PROGRAM F_VELOCIDADES
VAR_INPUT
	Func:E_Funcio;
END_VAR
VAR
	///Activa
	xActv: BOOL;
	///Parametros
	wP_SP_SpeedPumpC: WORD;
	wP_SP_Speed: WORD;
	wP_SP_T_Pass: WORD;
	///Fin Funcion
	xFinFunc: BOOL;
	tFinFuncion: Ton;
	a: INT;
	rOutAnalogSpeedPumpC: REAL;
END_VAR


a:=a+1;

(*Activa funcio *)
xActv:= func.Actv_Funcio;

wP_SP_SpeedPumpC:= func.ParamFunc[1];
wP_SP_Speed:= func.ParamFunc[2];
wP_SP_T_Pass:= func.ParamFunc[3];

(*
IF xActv
	THEN
	(*Torniquets*)
	IF wP_SP_Speed>0 THEN
		Mc.WINCH.iSP_Speed:=WORD_TO_INT(wP_SP_Speed);
	END_IF

	IF wP_SP_T_Pass>0 THEN
		Mc.WINCH.iSP_T_Pass:=WORD_TO_INT(wP_SP_T_Pass);
	END_IF
	*)

(*Bomba*)
IF wP_SP_SpeedPumpC >0 THEN
		mc._08_CIRC.rSP_SpeedPumpC:=  Canvi_Escala(
													In:= wP_SP_SpeedPumpC, 
													In_Min:= Mc._09_CPUMP.iPF_AnaMin_UF, 
													In_Max:= Mc._09_CPUMP.iPF_AnaMax_UF, 
													Out_Min:= 0, 
													Out_Max:= 100);
END_IF
	
		
(*Fin funcio *)
tFinFuncion(IN:=xActv , PT:=T#5S);
xFinFunc:= tFinFuncion.Q;

END_PROGRAM

(* stored: Version 1.1.0.1, ProductVersion 3.1.4024.10
   POU F_VELOCIDADES: Id {26e5b4cd-1fa4-47e9-ac1e-20319444c7ee}, SpecialFunc None *)
